TYPE ST_TransportControlParamEmulation :
(**************************************************************************************
 * 	Application		:	BoxControl Framework
 *	Revision		:	$Revision: 404529 $
 *	Revision date	:	$Date: 2018-04-23 08:21:38 +0200 (Mo., 23 Apr 2018) $
 *	Last changed by	:	$Author: b7bolm $
 *	URL				:	$URL: http://almscdc.swisslog.com/repo/SWPD/Development/BoxControlFramework/20_Release/trunk/01_Software/BCF/BCF/JumpStart/20_Product/11_Emu/12_E_Functions/10_Lib/10_Conv/01_DUTs/ST_TransportControlParamEmulation.TcDUT $
 *
 *	Purpose			:	Transport control parameter emulation
 *
 * ------------------------------------------------------------------------------------
 *	Copyright Swisslog [IP AG], Switzerland. All rights reserved.
 * 
 * ------------------------------------------------------------------------------------
 *	
 * 	Revision History: 
 *
 * 	VERSION			DATE			INITIALS			DESCRIPTION
 *	0.1				01.01.2001		swl					Example
 *
 **************************************************************************************)	
STRUCT
	eFunctionNumber			: E_FunctionNumber; // Number oft the function
	FunctionState			: ST_PositionState; // Function state
	ZoneNumber 				: INT; // Number of the zone
	Settings 				: ST_CFG_Zone; // Settings of the zone
	TransportParam          : ST_TransportParam; // Paramter of the current transport
	//ZoneEnable      		: ST_TransportEnable; // Zone enable
	//ExternalZoneEnable 		: BOOL; // External enable 
END_STRUCT
END_TYPE

(* stored: Version 1.1.0.1, ProductVersion 3.1.4022.18
   DUT ST_TransportControlParamEmulation: Id {eacf531c-7263-48af-b00b-9304f4f35417} *)
